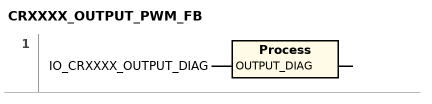
// NETWORK 1
Process(OUTPUT_DIAG := IO_CRXXXX_OUTPUT_DIAG);

METHOD PUBLIC Process
VAR_INPUT
END_VAR

VAR
	uiValue_Prev: UINT;
	uiValue_Changes: UINT;
	INIT_CDL: BOOL:=TRUE;
END_VAR

VAR_IN_OUT
	OUTPUT_DIAG: CRXXXX_OUTPUT_DATA;
END_VAR
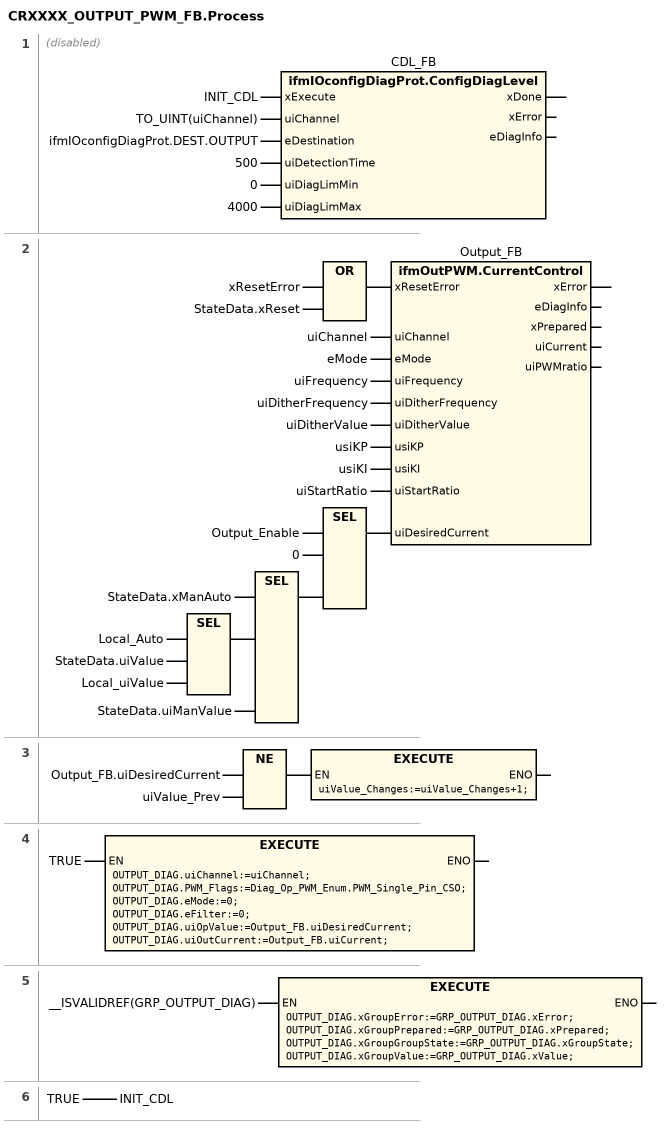
// NETWORK 1 (disabled)
// CDL_FB(
//     xExecute := INIT_CDL,
//     uiChannel := TO_UINT(uiChannel),
//     eDestination := ifmIOconfigDiagProt.DEST.OUTPUT,
//     uiDetectionTime := 500,
//     uiDiagLimMin := 0,
//     uiDiagLimMax := 4000); // ifmIOconfigDiagProt.ConfigDiagLevel

// NETWORK 2
Output_FB(
    xResetError := xResetError OR StateData.xReset,
    uiChannel := uiChannel,
    eMode := eMode,
    uiFrequency := uiFrequency,
    uiDitherFrequency := uiDitherFrequency,
    uiDitherValue := uiDitherValue,
    usiKP := usiKP,
    usiKI := usiKI,
    uiStartRatio := uiStartRatio,
    uiDesiredCurrent := SEL(Output_Enable, 0, SEL(StateData.xManAuto, SEL(Local_Auto, StateData.uiValue, Local_uiValue), StateData.uiManValue))); // ifmOutPWM.CurrentControl

// NETWORK 3
IF Output_FB.uiDesiredCurrent <> uiValue_Prev THEN uiValue_Changes:=uiValue_Changes+1; END_IF

// NETWORK 4
OUTPUT_DIAG.uiChannel:=uiChannel;
OUTPUT_DIAG.PWM_Flags:=Diag_Op_PWM_Enum.PWM_Single_Pin_CSO;
OUTPUT_DIAG.eMode:=0;
OUTPUT_DIAG.eFilter:=0;
OUTPUT_DIAG.uiOpValue:=Output_FB.uiDesiredCurrent;
OUTPUT_DIAG.uiOutCurrent:=Output_FB.uiCurrent;

// NETWORK 5
IF __ISVALIDREF(GRP_OUTPUT_DIAG) THEN
    OUTPUT_DIAG.xGroupError:=GRP_OUTPUT_DIAG.xError;
    OUTPUT_DIAG.xGroupPrepared:=GRP_OUTPUT_DIAG.xPrepared;
    OUTPUT_DIAG.xGroupGroupState:=GRP_OUTPUT_DIAG.xGroupState;
    OUTPUT_DIAG.xGroupValue:=GRP_OUTPUT_DIAG.xValue;
END_IF

// NETWORK 6
INIT_CDL := TRUE;
END_METHOD

END_FUNCTION_BLOCK

// StandardPLC/Application/App_PLC/PLC_PRG_APP
PROGRAM PLC_PRG_APP
VAR
END_VAR

END_PROGRAM

// Project Information/GetCompany
// This function has been automatically generated from the project information.
{attribute 'signature_flag' := '1073741824'}
{attribute 'register_in_runtime'}
FUNCTION GetCompany : WSTRING
VAR_INPUT
	
END_VAR

GetCompany := "Mtech";

END_FUNCTION

// Project Information/GetTitle
// This function has been automatically generated from the project information.
{attribute 'signature_flag' := '1073741824'}
{attribute 'register_in_runtime'}
FUNCTION GetTitle : WSTRING
VAR_INPUT
	
END_VAR

GetTitle := "T620X PLC";

END_FUNCTION

// Project Information/GetVersion
// This function has been automatically generated from the project information.
{attribute 'signature_flag' := '1073741824'}
{attribute 'register_in_runtime'}
FUNCTION GetVersion : VERSION
VAR_INPUT
	
END_VAR

GetVersion.uiMajor := 1;
GetVersion.uiMinor := 0;
GetVersion.uiServicePack := 3;
GetVersion.uiPatch := 0;

END_FUNCTION

// Project Information/GetTextProperty2
// This function has been automatically generated from the project information.
{attribute 'signature_flag' := '1073741824'}
{attribute 'register_in_runtime'}
FUNCTION GetTextProperty2 : POINTER TO WSTRING
VAR_INPUT
	stKey: WSTRING;
END_VAR

IF stKey = "Company" THEN
	GetTextProperty2 := ADR("Mtech");
ELSIF stKey = "Description" THEN
	GetTextProperty2 := ADR("");
ELSIF stKey = "Project" THEN
	GetTextProperty2 := ADR("T620X_PLC_CR711S_SP16p5_32bit");
ELSIF stKey = "Title" THEN
	GetTextProperty2 := ADR("T620X PLC");
ELSE
	GetTextProperty2 := ADR("");
END_IF

END_FUNCTION

// Project Information/GetNumberProperty
// This function has been automatically generated from the project information.
{attribute 'signature_flag' := '1073741824'}
{attribute 'register_in_runtime'}
FUNCTION GetNumberProperty : DINT
VAR_INPUT
	stKey: WSTRING;
END_VAR

GetNumberProperty := 0;

END_FUNCTION

// Project Information/GetVersionProperty
// This function has been automatically generated from the project information.
{attribute 'signature_flag' := '1073741824'}
{attribute 'register_in_runtime'}
FUNCTION GetVersionProperty : VERSION
VAR_INPUT
	stKey: WSTRING;
END_VAR

IF stKey = "Version" THEN
	GetVersionProperty.uiMajor := 1;
	GetVersionProperty.uiMinor := 0;
	GetVersionProperty.uiServicePack := 3;
	GetVersionProperty.uiPatch := 0;
ELSE
	GetVersionProperty.uiMajor := 0;
	GetVersionProperty.uiMinor := 0;
	GetVersionProperty.uiServicePack := 0;
	GetVersionProperty.uiPatch := 0;
END_IF

END_FUNCTION

// StandardPLC/Application/Visualisations/Input_IFM_PLC_CRXXXX
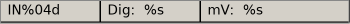
VISUALIZATION Input_IFM_PLC_CRXXXX  // 350x24
VAR_IN_OUT
	Input: CRXXXX_INPUT_DATA;
END_VAR
VAR
END_VAR
    Textfield (100,-2 100x24), "Dig: %s", text variable: Input.xValueDigital, colour toggle: Input.xValueDigital
    Textfield (200,-2 150x24), "mV: %s", text variable: Input.uiValueAnalogue
    Textfield (0,-2 100x24), "IN%04d", text variable: Input.uiChannel
END_VISUALIZATION

// StandardPLC/Application/Visualisations/Output_IFM_PLC_CRXXXX
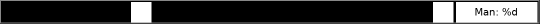
VISUALIZATION Output_IFM_PLC_CRXXXX  // 540x24
VAR_IN_OUT
	Output_States: CRXXXX_OUTPUT_STATE_DATA;	
	Output_Diag: CRXXXX_OUTPUT_DATA;
END_VAR
VAR
END_VAR
    Textfield (154,0 61x24), "%s mA", text variable: Output_Diag.uiOutCurrent
    Textfield (263,-1 163x24), "i: %s", text variable: Output_Diag.eDiagInfo
    Textfield (72,0 55x24), "Op:%d", text variable: Output_Diag.uiOpValue
    Textfield (0,0 70x24), "OUT%04d", text variable: Output_Diag.uiChannel
    Rectangle (131,2 20x20), colour toggle: Output_Diag.uiOpValue
    Rectangle (456,2 81x20), "Man: %d", text variable: Output_States.uiManValue, colour toggle: Output_States.uiManValue
        OnMouseClick: write the text variable via VisuDialogs.Numpad, min 0, max 1000
    Rectangle (433,2 20x20), colour toggle: Output_States.xManAuto
        toggle Output_States.xManAuto
    Textfield (219,0 41x24), "E: %d", text variable: Output_Diag.xError
END_VISUALIZATION

// StandardPLC/Application/Visualisations/Output_IFM_PLC_CRXXXX_GROUP
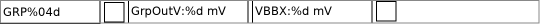
VISUALIZATION Output_IFM_PLC_CRXXXX_GROUP  // 540x24
VAR_IN_OUT
	Output_Diag: CRXXXX_OUTPUT_GROUP_DATA;
END_VAR
VAR
END_VAR
    Textfield (128,-1 120x24), "GrpOutV:%d mV", text variable: Output_Diag.uiGroupVoltage
    Textfield (0,0 100x24), "GRP%04d", text variable: Output_Diag.uiChannel
    Rectangle (376,1 20x20), colour toggle: Output_Diag.xGroupState
    Rectangle (104,2 20x20), colour toggle: Output_Diag.xError
    Textfield (252,-1 120x24), "VBBX:%d mV", text variable: Output_Diag.uiVBBxVoltage
END_VISUALIZATION

// StandardPLC/Application/Visualisations/Inputs_Test
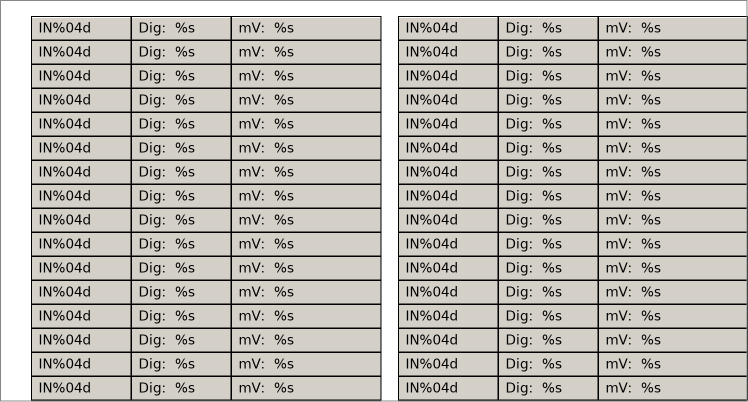
VISUALIZATION Inputs_Test  // 748x402
    Frame (31,18 350x24)
        shows Input_IFM_PLC_CRXXXX(Input := NVL_UDP_TX.All_Inputs.IN0100)
    Frame (31,42 350x24)
        shows Input_IFM_PLC_CRXXXX(Input := NVL_UDP_TX.All_Inputs.IN0101)
    Frame (31,66 350x24)
        shows Input_IFM_PLC_CRXXXX(Input := NVL_UDP_TX.All_Inputs.IN0102)
    Frame (31,90 350x24)
        shows Input_IFM_PLC_CRXXXX(Input := NVL_UDP_TX.All_Inputs.IN0103)
    Frame (31,114 350x24)
        shows Input_IFM_PLC_CRXXXX(Input := NVL_UDP_TX.All_Inputs.IN0200)
    Frame (31,138 350x24)
        shows Input_IFM_PLC_CRXXXX(Input := NVL_UDP_TX.All_Inputs.IN0201)
    Frame (31,162 350x24)
        shows Input_IFM_PLC_CRXXXX(Input := NVL_UDP_TX.All_Inputs.IN0202)
    Frame (31,186 350x24)
        shows Input_IFM_PLC_CRXXXX(Input := NVL_UDP_TX.All_Inputs.IN0203)
    Frame (31,210 350x24)
        shows Input_IFM_PLC_CRXXXX(Input := NVL_UDP_TX.All_Inputs.IN0600)
    Frame (31,234 350x24)
        shows Input_IFM_PLC_CRXXXX(Input := NVL_UDP_TX.All_Inputs.IN0601)
    Frame (31,258 350x24)
        shows Input_IFM_PLC_CRXXXX(Input := NVL_UDP_TX.All_Inputs.IN0602)
    Frame (31,282 350x24)
        shows Input_IFM_PLC_CRXXXX(Input := NVL_UDP_TX.All_Inputs.IN0603)
    Frame (31,306 350x24)
        shows Input_IFM_PLC_CRXXXX(Input := NVL_UDP_TX.All_Inputs.IN0700)
    Frame (31,330 350x24)
        shows Input_IFM_PLC_CRXXXX(Input := NVL_UDP_TX.All_Inputs.IN0701)
    Frame (31,354 350x24)
        shows Input_IFM_PLC_CRXXXX(Input := NVL_UDP_TX.All_Inputs.IN0702)
    Frame (31,378 350x24)
        shows Input_IFM_PLC_CRXXXX(Input := NVL_UDP_TX.All_Inputs.IN0703)
    Frame (398,18 350x24)
        shows Input_IFM_PLC_CRXXXX(Input := NVL_UDP_TX.All_Inputs.IN0000)
    Frame (398,42 350x24)
        shows Input_IFM_PLC_CRXXXX(Input := NVL_UDP_TX.All_Inputs.IN0001)
    Frame (398,66 350x24)
        shows Input_IFM_PLC_CRXXXX(Input := NVL_UDP_TX.All_Inputs.IN0002)
    Frame (398,90 350x24)
        shows Input_IFM_PLC_CRXXXX(Input := NVL_UDP_TX.All_Inputs.IN0003)
    Frame (398,114 350x24)
        shows Input_IFM_PLC_CRXXXX(Input := NVL_UDP_TX.All_Inputs.IN0500)
    Frame (398,138 350x24)
        shows Input_IFM_PLC_CRXXXX(Input := NVL_UDP_TX.All_Inputs.IN0501)
    Frame (398,162 350x24)
        shows Input_IFM_PLC_CRXXXX(Input := NVL_UDP_TX.All_Inputs.IN0502)
    Frame (398,186 350x24)
        shows Input_IFM_PLC_CRXXXX(Input := NVL_UDP_TX.All_Inputs.IN0503)
    Frame (398,210 350x24)
        shows Input_IFM_PLC_CRXXXX(Input := NVL_UDP_TX.All_Inputs.IN0400)
    Frame (398,234 350x24)
        shows Input_IFM_PLC_CRXXXX(Input := NVL_UDP_TX.All_Inputs.IN0401)
    Frame (398,258 350x24)
        shows Input_IFM_PLC_CRXXXX(Input := NVL_UDP_TX.All_Inputs.IN0900)
    Frame (398,282 350x24)
        shows Input_IFM_PLC_CRXXXX(Input := NVL_UDP_TX.All_Inputs.IN0901)
    Frame (398,306 350x24)
        shows Input_IFM_PLC_CRXXXX(Input := NVL_UDP_TX.All_Inputs.IN0300)
    Frame (398,330 350x24)
        shows Input_IFM_PLC_CRXXXX(Input := NVL_UDP_TX.All_Inputs.IN0301)
    Frame (398,354 350x24)
        shows Input_IFM_PLC_CRXXXX(Input := NVL_UDP_TX.All_Inputs.IN0800)
    Frame (398,378 350x24)
        shows Input_IFM_PLC_CRXXXX(Input := NVL_UDP_TX.All_Inputs.IN0801)
END_VISUALIZATION

// StandardPLC/Application/Visualisations/Outputs_Test
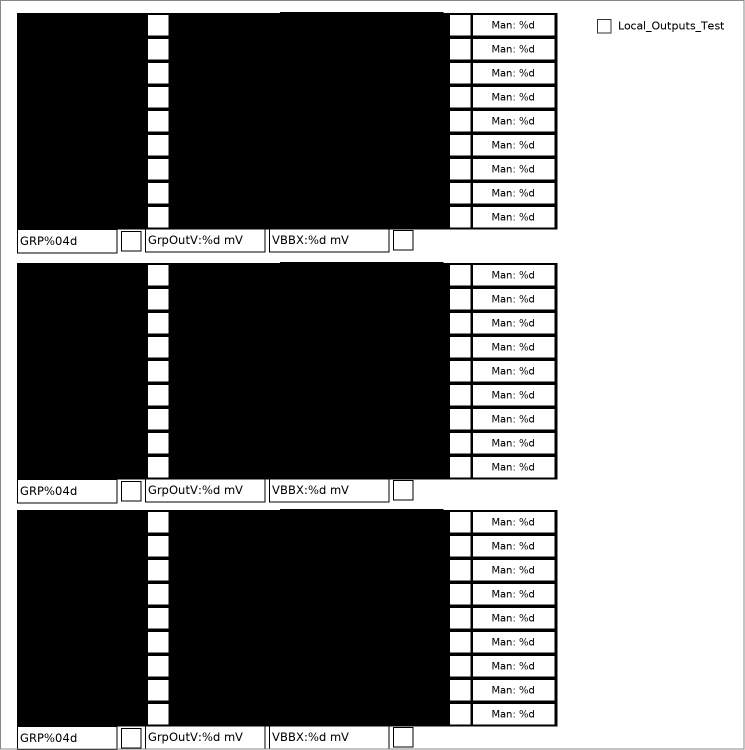
VISUALIZATION Outputs_Test  // 745x750
    Frame (17,13 540x24)
        shows Output_IFM_PLC_CRXXXX(Output_States := NVL_UDP_RX.All.OUT0000, Output_Diag := NVL_UDP_TX.All_Outputs_Diag.OUT0000)
    Frame (17,37 540x24)
        shows Output_IFM_PLC_CRXXXX(Output_States := NVL_UDP_RX.All.OUT0001, Output_Diag := NVL_UDP_TX.All_Outputs_Diag.OUT0001)
    Frame (17,61 540x24)
        shows Output_IFM_PLC_CRXXXX(Output_States := NVL_UDP_RX.All.OUT0002, Output_Diag := NVL_UDP_TX.All_Outputs_Diag.OUT0002)
    Frame (17,85 540x24)
        shows Output_IFM_PLC_CRXXXX(Output_States := NVL_UDP_RX.All.OUT0003, Output_Diag := NVL_UDP_TX.All_Outputs_Diag.OUT0003)
    Frame (17,109 540x24)
        shows Output_IFM_PLC_CRXXXX(Output_States := NVL_UDP_RX.All.OUT0004, Output_Diag := NVL_UDP_TX.All_Outputs_Diag.OUT0004)
    Frame (17,133 540x24)
        shows Output_IFM_PLC_CRXXXX(Output_States := NVL_UDP_RX.All.OUT0005, Output_Diag := NVL_UDP_TX.All_Outputs_Diag.OUT0005)
    Frame (17,157 540x24)
        shows Output_IFM_PLC_CRXXXX(Output_States := NVL_UDP_RX.All.OUT0006, Output_Diag := NVL_UDP_TX.All_Outputs_Diag.OUT0006)
    Frame (17,181 540x24)
        shows Output_IFM_PLC_CRXXXX(Output_States := NVL_UDP_RX.All.OUT0007, Output_Diag := NVL_UDP_TX.All_Outputs_Diag.OUT0007)
    Frame (17,205 540x24)
        shows Output_IFM_PLC_CRXXXX(Output_States := NVL_UDP_RX.All.OUT0008, Output_Diag := NVL_UDP_TX.All_Outputs_Diag.OUT0008)
    Frame (17,263 540x24)
        shows Output_IFM_PLC_CRXXXX(Output_States := NVL_UDP_RX.All.OUT0100, Output_Diag := NVL_UDP_TX.All_Outputs_Diag.OUT0100)
    Frame (17,287 540x24)
        shows Output_IFM_PLC_CRXXXX(Output_States := NVL_UDP_RX.All.OUT0101, Output_Diag := NVL_UDP_TX.All_Outputs_Diag.OUT0101)
    Frame (17,311 540x24)
        shows Output_IFM_PLC_CRXXXX(Output_States := NVL_UDP_RX.All.OUT0102, Output_Diag := NVL_UDP_TX.All_Outputs_Diag.OUT0102)
    Frame (17,335 540x24)
        shows Output_IFM_PLC_CRXXXX(Output_States := NVL_UDP_RX.All.OUT0103, Output_Diag := NVL_UDP_TX.All_Outputs_Diag.OUT0103)
    Frame (17,359 540x24)
        shows Output_IFM_PLC_CRXXXX(Output_States := NVL_UDP_RX.All.OUT0104, Output_Diag := NVL_UDP_TX.All_Outputs_Diag.OUT0104)
    Frame (17,383 540x24)
        shows Output_IFM_PLC_CRXXXX(Output_States := NVL_UDP_RX.All.OUT0105, Output_Diag := NVL_UDP_TX.All_Outputs_Diag.OUT0105)
    Frame (17,407 540x24)
        shows Output_IFM_PLC_CRXXXX(Output_States := NVL_UDP_RX.All.OUT0106, Output_Diag := NVL_UDP_TX.All_Outputs_Diag.OUT0106)
    Frame (17,431 540x24)
        shows Output_IFM_PLC_CRXXXX(Output_States := NVL_UDP_RX.All.OUT0107, Output_Diag := NVL_UDP_TX.All_Outputs_Diag.OUT0107)
    Frame (17,455 540x24)
        shows Output_IFM_PLC_CRXXXX(Output_States := NVL_UDP_RX.All.OUT0108, Output_Diag := NVL_UDP_TX.All_Outputs_Diag.OUT0108)
    Frame (17,510 540x24)
        shows Output_IFM_PLC_CRXXXX(Output_States := NVL_UDP_RX.All.OUT0200, Output_Diag := NVL_UDP_TX.All_Outputs_Diag.OUT0200)
    Frame (17,534 540x24)
        shows Output_IFM_PLC_CRXXXX(Output_States := NVL_UDP_RX.All.OUT0201, Output_Diag := NVL_UDP_TX.All_Outputs_Diag.OUT0201)
    Frame (17,558 540x24)
        shows Output_IFM_PLC_CRXXXX(Output_States := NVL_UDP_RX.All.OUT0202, Output_Diag := NVL_UDP_TX.All_Outputs_Diag.OUT0202)
    Frame (17,582 540x24)
        shows Output_IFM_PLC_CRXXXX(Output_States := NVL_UDP_RX.All.OUT0203, Output_Diag := NVL_UDP_TX.All_Outputs_Diag.OUT0203)
    Frame (17,606 540x24)
        shows Output_IFM_PLC_CRXXXX(Output_States := NVL_UDP_RX.All.OUT0204, Output_Diag := NVL_UDP_TX.All_Outputs_Diag.OUT0204)
    Frame (17,630 540x24)
        shows Output_IFM_PLC_CRXXXX(Output_States := NVL_UDP_RX.All.OUT0205, Output_Diag := NVL_UDP_TX.All_Outputs_Diag.OUT0205)
    Frame (17,654 540x24)
        shows Output_IFM_PLC_CRXXXX(Output_States := NVL_UDP_RX.All.OUT0206, Output_Diag := NVL_UDP_TX.All_Outputs_Diag.OUT0206)
    Frame (17,678 540x24)
        shows Output_IFM_PLC_CRXXXX(Output_States := NVL_UDP_RX.All.OUT0207, Output_Diag := NVL_UDP_TX.All_Outputs_Diag.OUT0207)
    Frame (17,702 540x24)
        shows Output_IFM_PLC_CRXXXX(Output_States := NVL_UDP_RX.All.OUT0208, Output_Diag := NVL_UDP_TX.All_Outputs_Diag.OUT0208)
    Checkbox (595,11 150x30), "Local_Outputs_Test", variable: PLC_UDP_WDT_Check.Local_Outputs_Test
    Frame (17,229 540x24)
        shows Output_IFM_PLC_CRXXXX_GROUP(Output_Diag := NVL_UDP_TX.All_Outputs_Diag.GROUP0)
    Frame (17,479 540x24)
        shows Output_IFM_PLC_CRXXXX_GROUP(Output_Diag := NVL_UDP_TX.All_Outputs_Diag.GROUP1)
    Frame (17,726 540x24)
        shows Output_IFM_PLC_CRXXXX_GROUP(Output_Diag := NVL_UDP_TX.All_Outputs_Diag.GROUP2)
END_VISUALIZATION
